Universal Robots PolyScope program: rtde_streaming_control_loop.urp

Program rtde_streaming_control_loop (installation=default directory=/ursim/programs createdIn=5.24.0 lastSavedIn=5.24.0 robotSerialNumber=20195599999)
Calibrated DH parameters: a=[0, -0.425, -0.3922, 0, 0, 0]; d=[0.1625, 0, 0, 0.1333, 0.0997, 0.0996]; alpha=[1.570796, 0, 0, 1.570796, -1.570796, 0]; deltaTheta=[0, 0, 0, 0, 0, 0]
InitVariablesNode
BeforeStart
  Script: rtde_set_watchdog("input_int_register_0", 1, "PAUSE")
  setp := get_actual_tcp_pose()
Robot Program (runOnlyOnce=false)
  Loop Forever
    Script file /ursim/programs/servoj_movement_sync.script
      | servoj(get_inverse_kin(setp, get_actual_joint_positions()), 0, 0, 0.008, 0.1, 300)
      | sync()
Thread Thread_1 (runOnlyOnce=false)
  Loop Forever
    Script file /ursim/programs/input_register_thread.script
      | global tmp = p[0,0,0,0,0,0]
      | tmp[0] = read_input_float_register(0)
      | tmp[1] = read_input_float_register(1)
      | tmp[2] = read_input_float_register(2)
      | tmp[3] = read_input_float_register(3)
      | tmp[4] = read_input_float_register(4)
      | tmp[5] = read_input_float_register(5)
      | setp = tmp
      | sync()
